# EPICS autosave request: gardasoftLED/PP400SeriesChannel_settings.req
$(P):CH$(CHANNEL):DESCRIPTION
